{attribute 'no-analysis'}
TYPE ST_VerificationResult :
STRUCT
	hr 		: HRESULT;
	sDiff 	: STRING(Param_TcHaxx_Snappy.cSnappyVerificationResultLength);
END_STRUCT
END_TYPE

(* stored: Version 1.1.0.1, ProductVersion 3.1.4026.18
   DUT ST_VerificationResult: Id {b0c070fc-92f1-4738-82f4-d2b7ebd9b938} *)
